FUNCTION_BLOCK FB_AxisReadNC
VAR_INPUT
	bExecute: BOOL;
	bReset: BOOL;
END_VAR
VAR_IN_OUT
	stConfig: ST_AxisParams;
	Axis: AXIS_REF;
END_VAR
VAR_OUTPUT
	bValid: BOOL;
	bBusy: BOOL;
	bError: BOOL;
	nErrorID: UDINT;
END_VAR
VAR
	iCycles: INT := 0;
	bReadOk: BOOL := FALSE;
	bInnerExec: BOOL := FALSE;
	fbReadRefVel: MC_ReadParameter;
  	fbReadRefVelRisingEdge: R_TRIG;
	fbReadMaxVel: MC_ReadParameter;
  	fbReadMaxVelRisingEdge: R_TRIG;
	fbReadMaxAcc: MC_ReadParameter;
  	fbReadMaxAccRisingEdge: R_TRIG;
	fbReadMaxDec: MC_ReadParameter;
  	fbReadMaxDecRisingEdge: R_TRIG;
	fbReadDefAcc: MC_ReadParameter;
  	fbReadDefAccRisingEdge: R_TRIG;
	fbReadDefDec: MC_ReadParameter;
  	fbReadDefDecRisingEdge: R_TRIG;
	fbReadDefJerk: MC_ReadParameter;
  	fbReadDefJerkRisingEdge: R_TRIG;
	fbReadHomeSearch: MC_ReadParameter;
  	fbReadHomeSearchRisingEdge: R_TRIG;
	fbReadHomeSync: MC_ReadParameter;
  	fbReadHomeSyncRisingEdge: R_TRIG;
	fbReadManFast: MC_ReadParameter;
  	fbReadManFastRisingEdge: R_TRIG;
	fbReadManSlow: MC_ReadParameter;
  	fbReadManSlowRisingEdge: R_TRIG;
	fbReadDeadTime: MC_ReadParameter;
  	fbReadDeadTimeRisingEdge: R_TRIG;
	fbReadEncScale: MC_ReadParameter;
  	fbReadEncScaleRisingEdge: R_TRIG;
	fbReadEncInvert: MC_ReadBoolParameter;
  	fbReadEncInvertRisingEdge: R_TRIG;
	fbReadMotInvert: MC_ReadBoolParameter;
  	fbReadMotInvertRisingEdge: R_TRIG;
END_VAR

// File auto-generated! Take care editing!
// Clears errors and allows a new read
IF bReset THEN
	bExecute := FALSE;
	bReset := FALSE;
END_IF
// Fails in the first n cycles depending on terminals, wait a bit
IF NOT bReadOk THEN
	iCycles := iCycles + 1;
	IF iCycles > 100 THEN
		bReadOk := TRUE;
	END_IF
END_IF
bInnerExec := bExecute AND bReadOk;
fbReadRefVel(Enable:=bInnerExec,
	ParameterNumber:=MC_AxisParameter.AxisRefVeloOnRefOutput,
	ReadMode:=E_ReadMode.READMODE_ONCE,
	Axis:=Axis);
fbReadRefVelRisingEdge(CLK:=fbReadRefVel.Valid AND NOT fbReadRefVel.Busy);
IF fbReadRefVelRisingEdge.Q AND NOT fbReadRefVel.Error THEN
	stConfig.ref_vel := fbReadRefVel.Value;
END_IF
fbReadMaxVel(Enable:=bInnerExec,
	ParameterNumber:=MC_AxisParameter.AxisMaxVelocity,
	ReadMode:=E_ReadMode.READMODE_ONCE,
	Axis:=Axis);
fbReadMaxVelRisingEdge(CLK:=fbReadMaxVel.Valid AND NOT fbReadMaxVel.Busy);
IF fbReadMaxVelRisingEdge.Q AND NOT fbReadMaxVel.Error THEN
	stConfig.max_vel := fbReadMaxVel.Value;
END_IF
fbReadMaxAcc(Enable:=bInnerExec,
	ParameterNumber:=MC_AxisParameter.MaxAccelerationSystem,
	ReadMode:=E_ReadMode.READMODE_ONCE,
	Axis:=Axis);
fbReadMaxAccRisingEdge(CLK:=fbReadMaxAcc.Valid AND NOT fbReadMaxAcc.Busy);
IF fbReadMaxAccRisingEdge.Q AND NOT fbReadMaxAcc.Error THEN
	stConfig.max_acc := fbReadMaxAcc.Value;
END_IF
fbReadMaxDec(Enable:=bInnerExec,
	ParameterNumber:=MC_AxisParameter.MaxDecelerationSystem,
	ReadMode:=E_ReadMode.READMODE_ONCE,
	Axis:=Axis);
fbReadMaxDecRisingEdge(CLK:=fbReadMaxDec.Valid AND NOT fbReadMaxDec.Busy);
IF fbReadMaxDecRisingEdge.Q AND NOT fbReadMaxDec.Error THEN
	stConfig.max_dec := fbReadMaxDec.Value;
END_IF
fbReadDefAcc(Enable:=bInnerExec,
	ParameterNumber:=MC_AxisParameter.AxisAcc,
	ReadMode:=E_ReadMode.READMODE_ONCE,
	Axis:=Axis);
fbReadDefAccRisingEdge(CLK:=fbReadDefAcc.Valid AND NOT fbReadDefAcc.Busy);
IF fbReadDefAccRisingEdge.Q AND NOT fbReadDefAcc.Error THEN
	stConfig.def_acc := fbReadDefAcc.Value;
END_IF
fbReadDefDec(Enable:=bInnerExec,
	ParameterNumber:=MC_AxisParameter.AxisDec,
	ReadMode:=E_ReadMode.READMODE_ONCE,
	Axis:=Axis);
fbReadDefDecRisingEdge(CLK:=fbReadDefDec.Valid AND NOT fbReadDefDec.Busy);
IF fbReadDefDecRisingEdge.Q AND NOT fbReadDefDec.Error THEN
	stConfig.def_dec := fbReadDefDec.Value;
END_IF
fbReadDefJerk(Enable:=bInnerExec,
	ParameterNumber:=MC_AxisParameter.AxisJerk,
	ReadMode:=E_ReadMode.READMODE_ONCE,
	Axis:=Axis);
fbReadDefJerkRisingEdge(CLK:=fbReadDefJerk.Valid AND NOT fbReadDefJerk.Busy);
IF fbReadDefJerkRisingEdge.Q AND NOT fbReadDefJerk.Error THEN
	stConfig.def_jerk := fbReadDefJerk.Value;
END_IF
fbReadHomeSearch(Enable:=bInnerExec,
	ParameterNumber:=MC_AxisParameter.AxisCalibrationVelocityForward,
	ReadMode:=E_ReadMode.READMODE_ONCE,
	Axis:=Axis);
fbReadHomeSearchRisingEdge(CLK:=fbReadHomeSearch.Valid AND NOT fbReadHomeSearch.Busy);
IF fbReadHomeSearchRisingEdge.Q AND NOT fbReadHomeSearch.Error THEN
	stConfig.home_search := fbReadHomeSearch.Value;
END_IF
fbReadHomeSync(Enable:=bInnerExec,
	ParameterNumber:=MC_AxisParameter.AxisCalibrationVelocityBackward,
	ReadMode:=E_ReadMode.READMODE_ONCE,
	Axis:=Axis);
fbReadHomeSyncRisingEdge(CLK:=fbReadHomeSync.Valid AND NOT fbReadHomeSync.Busy);
IF fbReadHomeSyncRisingEdge.Q AND NOT fbReadHomeSync.Error THEN
	stConfig.home_sync := fbReadHomeSync.Value;
END_IF
fbReadManFast(Enable:=bInnerExec,
	ParameterNumber:=MC_AxisParameter.AxisManualVelocityFast,
	ReadMode:=E_ReadMode.READMODE_ONCE,
	Axis:=Axis);
fbReadManFastRisingEdge(CLK:=fbReadManFast.Valid AND NOT fbReadManFast.Busy);
IF fbReadManFastRisingEdge.Q AND NOT fbReadManFast.Error THEN
	stConfig.man_fast := fbReadManFast.Value;
END_IF
fbReadManSlow(Enable:=bInnerExec,
	ParameterNumber:=MC_AxisParameter.AxisManualVelocitySlow,
	ReadMode:=E_ReadMode.READMODE_ONCE,
	Axis:=Axis);
fbReadManSlowRisingEdge(CLK:=fbReadManSlow.Valid AND NOT fbReadManSlow.Busy);
IF fbReadManSlowRisingEdge.Q AND NOT fbReadManSlow.Error THEN
	stConfig.man_slow := fbReadManSlow.Value;
END_IF
fbReadDeadTime(Enable:=bInnerExec,
	ParameterNumber:=MC_AxisParameter.AxisDelayTimeVeloPosition,
	ReadMode:=E_ReadMode.READMODE_ONCE,
	Axis:=Axis);
fbReadDeadTimeRisingEdge(CLK:=fbReadDeadTime.Valid AND NOT fbReadDeadTime.Busy);
IF fbReadDeadTimeRisingEdge.Q AND NOT fbReadDeadTime.Error THEN
	stConfig.dead_time := fbReadDeadTime.Value;
END_IF
fbReadEncScale(Enable:=bInnerExec,
	ParameterNumber:=MC_AxisParameter.AxisEncoderScalingFactor,
	ReadMode:=E_ReadMode.READMODE_ONCE,
	Axis:=Axis);
fbReadEncScaleRisingEdge(CLK:=fbReadEncScale.Valid AND NOT fbReadEncScale.Busy);
IF fbReadEncScaleRisingEdge.Q AND NOT fbReadEncScale.Error THEN
	stConfig.enc_scale := fbReadEncScale.Value;
END_IF
fbReadEncInvert(Enable:=bInnerExec,
	ParameterNumber:=MC_AxisParameter.AxisEncoderDirectionInverse,
	ReadMode:=E_ReadMode.READMODE_ONCE,
	Axis:=Axis);
fbReadEncInvertRisingEdge(CLK:=fbReadEncInvert.Valid AND NOT fbReadEncInvert.Busy);
IF fbReadEncInvertRisingEdge.Q AND NOT fbReadEncInvert.Error THEN
	stConfig.enc_invert := fbReadEncInvert.Value;
END_IF
fbReadMotInvert(Enable:=bInnerExec,
	ParameterNumber:=MC_AxisParameter.AxisMotorDirectionInverse,
	ReadMode:=E_ReadMode.READMODE_ONCE,
	Axis:=Axis);
fbReadMotInvertRisingEdge(CLK:=fbReadMotInvert.Valid AND NOT fbReadMotInvert.Busy);
IF fbReadMotInvertRisingEdge.Q AND NOT fbReadMotInvert.Error THEN
	stConfig.mot_invert := fbReadMotInvert.Value;
END_IF
bValid := fbReadRefVel.Valid AND fbReadMaxVel.Valid AND fbReadMaxAcc.Valid AND fbReadMaxDec.Valid AND fbReadDefAcc.Valid AND fbReadDefDec.Valid AND fbReadDefJerk.Valid AND fbReadHomeSearch.Valid AND fbReadHomeSync.Valid AND fbReadManFast.Valid AND fbReadManSlow.Valid AND fbReadDeadTime.Valid AND fbReadEncScale.Valid AND fbReadEncInvert.Valid AND fbReadMotInvert.Valid;
bBusy := fbReadRefVel.Busy OR fbReadMaxVel.Busy OR fbReadMaxAcc.Busy OR fbReadMaxDec.Busy OR fbReadDefAcc.Busy OR fbReadDefDec.Busy OR fbReadDefJerk.Busy OR fbReadHomeSearch.Busy OR fbReadHomeSync.Busy OR fbReadManFast.Busy OR fbReadManSlow.Busy OR fbReadDeadTime.Busy OR fbReadEncScale.Busy OR fbReadEncInvert.Busy OR fbReadMotInvert.Busy;
bError := fbReadRefVel.Error OR fbReadMaxVel.Error OR fbReadMaxAcc.Error OR fbReadMaxDec.Error OR fbReadDefAcc.Error OR fbReadDefDec.Error OR fbReadDefJerk.Error OR fbReadHomeSearch.Error OR fbReadHomeSync.Error OR fbReadManFast.Error OR fbReadManSlow.Error OR fbReadDeadTime.Error OR fbReadEncScale.Error OR fbReadEncInvert.Error OR fbReadMotInvert.Error;
IF NOT bError THEN
	nErrorID := 0;
ELSIF fbReadRefVel.ErrorID > 0 THEN
	nErrorID := fbReadRefVel.ErrorID;
ELSIF fbReadMaxVel.ErrorID > 0 THEN
	nErrorID := fbReadMaxVel.ErrorID;
ELSIF fbReadMaxAcc.ErrorID > 0 THEN
	nErrorID := fbReadMaxAcc.ErrorID;
ELSIF fbReadMaxDec.ErrorID > 0 THEN
	nErrorID := fbReadMaxDec.ErrorID;
ELSIF fbReadDefAcc.ErrorID > 0 THEN
	nErrorID := fbReadDefAcc.ErrorID;
ELSIF fbReadDefDec.ErrorID > 0 THEN
	nErrorID := fbReadDefDec.ErrorID;
ELSIF fbReadDefJerk.ErrorID > 0 THEN
	nErrorID := fbReadDefJerk.ErrorID;
ELSIF fbReadHomeSearch.ErrorID > 0 THEN
	nErrorID := fbReadHomeSearch.ErrorID;
ELSIF fbReadHomeSync.ErrorID > 0 THEN
	nErrorID := fbReadHomeSync.ErrorID;
ELSIF fbReadManFast.ErrorID > 0 THEN
	nErrorID := fbReadManFast.ErrorID;
ELSIF fbReadManSlow.ErrorID > 0 THEN
	nErrorID := fbReadManSlow.ErrorID;
ELSIF fbReadDeadTime.ErrorID > 0 THEN
	nErrorID := fbReadDeadTime.ErrorID;
ELSIF fbReadEncScale.ErrorID > 0 THEN
	nErrorID := fbReadEncScale.ErrorID;
ELSIF fbReadEncInvert.ErrorID > 0 THEN
	nErrorID := fbReadEncInvert.ErrorID;
ELSIF fbReadMotInvert.ErrorID > 0 THEN
	nErrorID := fbReadMotInvert.ErrorID;
END_IF

END_FUNCTION_BLOCK

(* stored: Version 1.1.0.1, ProductVersion 3.1.4020.12
   POU FB_AxisReadNC: Id {ae0d0d38-2171-41e5-b49c-714adaf92c76}, SpecialFunc None *)
